PROGRAM MAIN
VAR
	LastMotorPosition	: 	UINT;
	Difference			:	INT;
	DrehzahlRpm			: 	REAL;
	DrehzahlRps			: 	REAL;
	OverflowCalculated	: 	BOOL := FALSE;
	UnderflowCalculated	: 	BOOL := FALSE;
END_VAR
VAR CONSTANT
	cycleTimeS			:	REAL := 0.01;
	ImpulsePerRevolution: 	UINT := 2048; 
	uintUpperBound		: 	UINT := 65535;
END_VAR


// calculate drehzahl
Difference := UINT_TO_INT(GVL_MOTOR.MotorPosition-LastMotorPosition);
// handle overflow / underflow
IF GVL_MOTOR.CounterOverflow AND OverflowCalculated = FALSE THEN
	OverflowCalculated := TRUE;
	Difference := UINT_TO_INT((uintUpperBound - LastMotorPosition) + GVL_MOTOR.MotorPosition);
ELSIF GVL_MOTOR.CounterOverflow = FALSE THEN   // reset flag
	OverflowCalculated := FALSE;
END_IF
IF GVL_MOTOR.CounterUnderflow AND UnderflowCalculated = FALSE THEN
	UnderflowCalculated := TRUE;
	Difference := UINT_TO_INT((GVL_MOTOR.MotorPosition - uintUpperBound) - LastMotorPosition);
ELSIF GVL_MOTOR.CounterUnderflow = FALSE THEN   // reset flag
	UnderflowCalculated := FALSE;
END_IF

DrehzahlRps := Difference / (cycleTimeS * ImpulsePerRevolution);
DrehzahlRpm := DrehzahlRps / 60;

// store values
LastMotorPosition := GVL_MOTOR.MotorPosition;

END_PROGRAM

(* stored: Version 1.1.0.1, ProductVersion 3.1.4024.9
   POU MAIN: Id {92c37176-988a-4ad3-8fd4-29743153aa41}, SpecialFunc None *)
